TYPE ST_PAOut_Valve :
STRUCT
	stMTOOutputs1:			ST_MTO_Outputs;
	stDoxControl1:			ST_DOX_Control;
	
	
	
END_STRUCT
END_TYPE

(* stored: Version 1.1.0.1, ProductVersion 3.1.4019.2
   DUT ST_PAOut_Valve: Id {36902021-48d3-4bef-9b24-0bfad59ff62e} *)
